PROGRAM PRG_InitializeControl
VAR
END_VAR

(* ---------------------------------------------------------
   程序骨架：设备初始化子状态机。
   所属任务：Task_CffMain，调用顺序5。
   唯一Owner：PRG_InitializeControl。
   当前阶段：不运动、不复位实际驱动、不伪造初始化完成。
   后续实现：Entry、Action、Success、Timeout和Fault。
   --------------------------------------------------------- *)

END_PROGRAM

(* stored: Version 1.1.0.1
   POU PRG_InitializeControl: Id {A2000000-0000-4000-8000-000000000009} *)
